Omron CX-Programmer project NewProject (CX-Programmer 9.61)

# PLC NewPLC1: CP1E E20

## Global symbols (name address type ; comment)
0.00 BOOL  ; UP
0.01 BOOL  ; DOWN
0.02 BOOL  ; RESET
10.02 BOOL  ; LAMPU1

## Program NewProgram1 (cyclic task 0)
Local symbols
U CHANNEL

### Section Section1

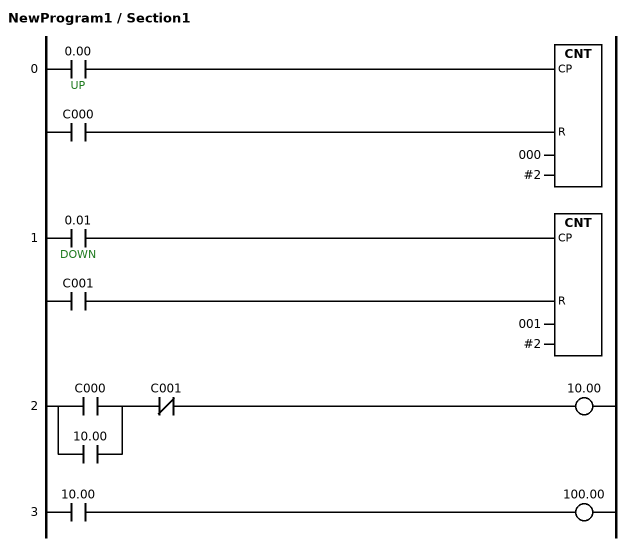
; rung 0
LD 0.00  ; UP
LD C000
CNT 000 #2
; rung 1
LD 0.01  ; DOWN
LD C001
CNT 001 #2
; rung 2
LD C000
OR 10.00
ANDNOT C001
OUT 10.00
; rung 3
LD 10.00
OUT 100.00

### Section END
; rung 0
END(001)